PROGRAM MAIN
VAR
END_VAR

END_PROGRAM

(* stored: Version 1.1.0.1
   POU MAIN: Id {2ac4e9c4-03fe-4954-80ea-bbc9e64ee4da} *)
